// TIA Portal project "BT2_B3_dengiaothong" (V14)

(* hardware
DEVICE "S7-1200 station_1"  S7-1200 Station
   slot 0: "Rack_0"  S7-1200 Rack  Rack  V1.0
   slot 1: "PLC_1"  CPU 1214C DC/DC/DC  6ES7 214-1AG40-0XB0  V4.2
*)

// ===== PLC "PLC_1"  CPU 1214C DC/DC/DC =====

VAR_GLOBAL   // PLC tag table "Default tag table"
   "UT1" AT %I0.0 : Bool;
   "Tag_1" AT %M0.0 : Bool;
   "X1" AT %Q0.0 : Bool;
   "D2" AT %Q0.1 : Bool;
   "UT2" AT %I0.1 : Bool;
   "D1" AT %Q0.2 : Bool;
   "X2" AT %Q0.3 : Bool;
   "Tag_4" AT %M0.1 : Bool;
   "CT_V" AT %I0.2 : Bool;
   "V1" AT %Q0.4 : Bool;
   "V2" AT %Q0.5 : Bool;
END_VAR

// folder: System blocks/Program resources

DATA_BLOCK "IEC_Timer_0_DB"   // DB1
{ S7_Optimized_Access := 'TRUE' }
AUTHOR : Simatic
FAMILY : IEC
NAME : IEC_TMR
VERSION : 1.0
// stored: InstanceOfName IEC_TIMER
"IEC_TIMER"
BEGIN
END_DATA_BLOCK

DATA_BLOCK "IEC_Timer_0_DB_1"   // DB2
{ S7_Optimized_Access := 'TRUE' }
AUTHOR : Simatic
FAMILY : IEC
NAME : IEC_TMR
VERSION : 1.0
// stored: InstanceOfName IEC_TIMER
"IEC_TIMER"
BEGIN
END_DATA_BLOCK

DATA_BLOCK "IEC_Timer_0_DB_2"   // DB3
{ S7_Optimized_Access := 'TRUE' }
AUTHOR : Simatic
FAMILY : IEC
NAME : IEC_TMR
VERSION : 1.0
// stored: InstanceOfName IEC_TIMER
"IEC_TIMER"
BEGIN
END_DATA_BLOCK

DATA_BLOCK "IEC_Timer_0_DB_3"   // DB4
{ S7_Optimized_Access := 'TRUE' }
AUTHOR : Simatic
FAMILY : IEC
NAME : IEC_TMR
VERSION : 1.0
// stored: InstanceOfName IEC_TIMER
"IEC_TIMER"
BEGIN
END_DATA_BLOCK

DATA_BLOCK "IEC_Timer_0_DB_4"   // DB5
{ S7_Optimized_Access := 'TRUE' }
AUTHOR : Simatic
FAMILY : IEC
NAME : IEC_TMR
VERSION : 1.0
// stored: InstanceOfName IEC_TIMER
"IEC_TIMER"
BEGIN
END_DATA_BLOCK

DATA_BLOCK "IEC_Timer_0_DB_5"   // DB6
{ S7_Optimized_Access := 'TRUE' }
AUTHOR : Simatic
FAMILY : IEC
NAME : IEC_TMR
VERSION : 1.0
// stored: InstanceOfName IEC_TIMER
"IEC_TIMER"
BEGIN
END_DATA_BLOCK

// folder: (top level)

ORGANIZATION_BLOCK "Main"   // OB1, LAD, ProgramCycle
TITLE = "Main Program Sweep (Cycle)"
{ S7_Optimized_Access := 'TRUE' }
VERSION : 0.1
   VAR_INPUT
      Initial_Call : Bool;   // Initial call of this OB
      Remanence : Bool;   // =True, if remanent data are available
   END_VAR
   VAR_TEMP   // added for the SCL form of the ladder/FBD networks
      _w1 : Bool;
   END_VAR
BEGIN

REGION Network 1
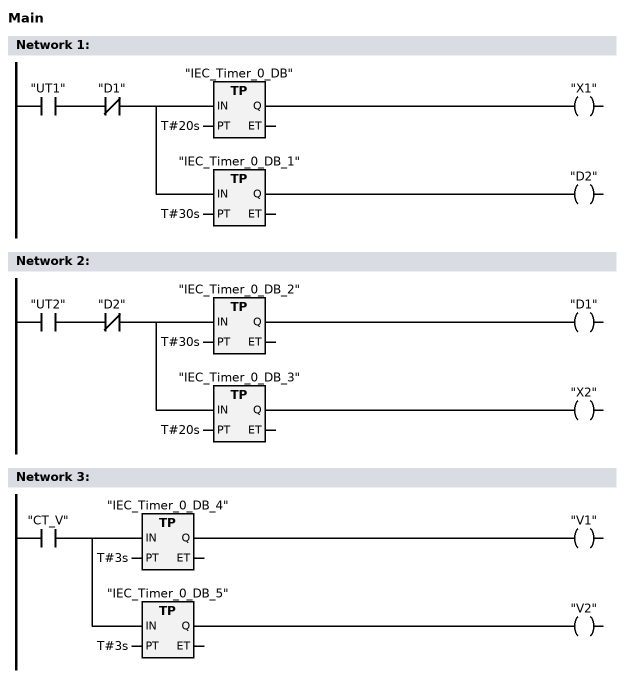
   #_w1 := "UT1" AND NOT "D1";
   "IEC_Timer_0_DB".TP(IN := #_w1, PT := T#20s);
   "X1" := "IEC_Timer_0_DB".Q;
   "IEC_Timer_0_DB_1".TP(IN := #_w1, PT := T#30s);
   "D2" := "IEC_Timer_0_DB_1".Q;
END_REGION

REGION Network 2
   #_w1 := "UT2" AND NOT "D2";
   "IEC_Timer_0_DB_2".TP(IN := #_w1, PT := T#30s);
   "D1" := "IEC_Timer_0_DB_2".Q;
   "IEC_Timer_0_DB_3".TP(IN := #_w1, PT := T#20s);
   "X2" := "IEC_Timer_0_DB_3".Q;
END_REGION

REGION Network 3
   "IEC_Timer_0_DB_4".TP(IN := "CT_V", PT := T#3s);
   "V1" := "IEC_Timer_0_DB_4".Q;
   "IEC_Timer_0_DB_5".TP(IN := "CT_V", PT := T#3s);
   "V2" := "IEC_Timer_0_DB_5".Q;
END_REGION
END_ORGANIZATION_BLOCK